// TwinCAT 3 PLC project PLC
// ProgramVersion: 3.1.4024.0
// libraries:
//   Tc2_Standard, * (Beckhoff Automation GmbH)
//   Tc2_System, * (Beckhoff Automation GmbH)
//   Tc3_Module, * (Beckhoff Automation GmbH)
// project tree:
//   / GlobalTextList.TcGTLO, PlcTask.TcTTO, Visualization Manager.TcVMO (not stored)
//   POUs/ MAIN.TcPOU
//   VISUs/ Visualization.TcVIS
// real-time tasks:
//   TASK PlcTask: cycle T#10ms, priority 20, ADS port 350

CONFIGURATION PLC
    RESOURCE PLC ON TwinCAT3
        TASK PlcTask(INTERVAL := T#10ms, PRIORITY := 20);
        PROGRAM MAIN WITH PlcTask : MAIN;
    END_RESOURCE
END_CONFIGURATION

// ---- POUs/MAIN.TcPOU
PROGRAM MAIN
VAR
	// push buttons
	StartPB: BOOL;
	StopPB: BOOL;
	ResetButton: BOOL;

	// sensors
	BottomLimitSwitch: BOOL;	
	ProxSwitch: BOOL;
	
	PistonLeftPos: BOOL;
	PistonRightPos: BOOL;
	
	// HW outputs
	
	ConveyorRun: BOOL;
	LifterUp: BOOL;
	LifterDown: BOOL;
	LifterStop: BOOL;
	
	PistonMoveLeft: BOOL;
	PistonMoveRight: BOOL;

	// Aux. objects
	rtBottomLS: R_TRIG;
	rtIndexPcb: R_TRIG;
	
	tondelayLifterUp: TON;
	tonDelay1sec: TON;
	
	rtPistonLeftReached: R_TRIG;
	ctuPistonLeftMovements: CTU;
END_VAR
VAR // added by the converter: edge detectors and wires of the graphical bodies
    _w1 : BOOL;
END_VAR

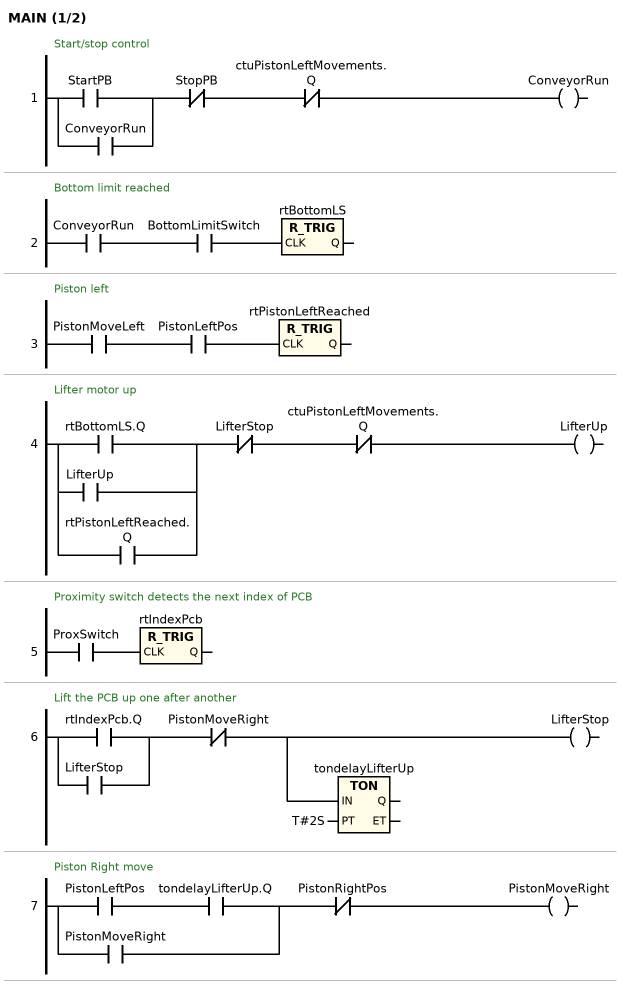
// NETWORK 1
// Start/stop control
ConveyorRun := (StartPB OR ConveyorRun) AND NOT StopPB AND NOT ctuPistonLeftMovements.Q;

// NETWORK 2
// Bottom limit reached
rtBottomLS(CLK := ConveyorRun AND BottomLimitSwitch); // R_TRIG

// NETWORK 3
// Piston left
rtPistonLeftReached(CLK := PistonMoveLeft AND PistonLeftPos); // R_TRIG

// NETWORK 4
// Lifter motor up
LifterUp := (rtBottomLS.Q OR LifterUp OR rtPistonLeftReached.Q) AND NOT LifterStop AND NOT ctuPistonLeftMovements.Q;

// NETWORK 5
// Proximity switch detects the next index of PCB
rtIndexPcb(CLK := ProxSwitch); // R_TRIG

// NETWORK 6
// Lift the PCB up one after another
_w1 := (rtIndexPcb.Q OR LifterStop) AND NOT PistonMoveRight;
LifterStop := _w1;
tondelayLifterUp(IN := _w1, PT := T#2S); // TON

// NETWORK 7
// Piston Right move
PistonMoveRight := (PistonLeftPos AND tondelayLifterUp.Q OR PistonMoveRight) AND NOT PistonRightPos;

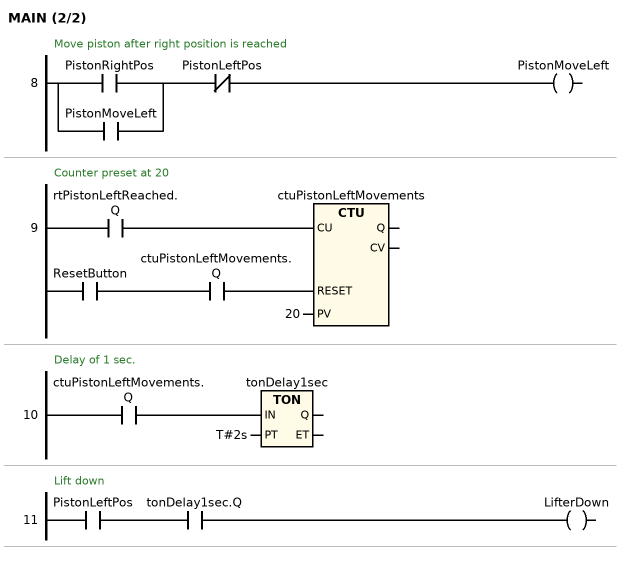
// NETWORK 8
// Move piston after right position is reached
PistonMoveLeft := (PistonRightPos OR PistonMoveLeft) AND NOT PistonLeftPos;

// NETWORK 9
// Counter preset at 20
ctuPistonLeftMovements(
    CU := rtPistonLeftReached.Q,
    RESET := ResetButton AND ctuPistonLeftMovements.Q,
    PV := 20); // CTU

// NETWORK 10
// Delay of 1 sec.
tonDelay1sec(IN := ctuPistonLeftMovements.Q, PT := T#2s); // TON

// NETWORK 11
// Lift down
LifterDown := PistonLeftPos AND tonDelay1sec.Q;

END_PROGRAM

// ---- GlobalTextList.TcGTLO
TEXTLIST GlobalTextList
  290 = 'Bottom LS'
  452 = 'Conveyor Run'
  528 = 'Lifter'
  534 = 'Piston Left Pos'
  221 = 'Piston Right Pos'
  535 = 'Prox. switch'
  58 = 'start PB'
  407 = 'stop PB'
  340 = 'stopPB'
END_TEXTLIST

// ---- VISUs/Visualization.TcVIS
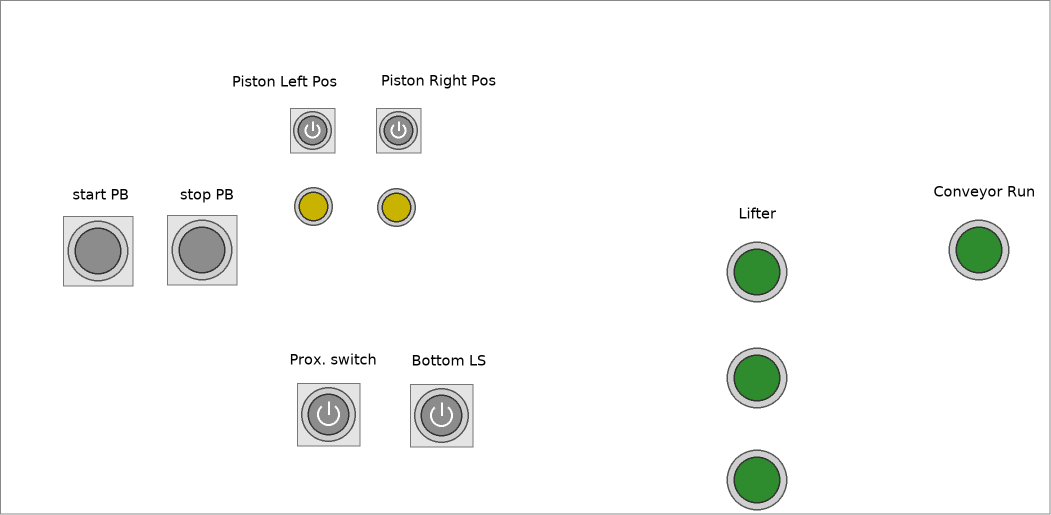
VISUALIZATION Visualization  // 1051x515
    PushSwitch (63,216 70x70), variable: MAIN.StartPB, behaviour: TAP, style: Switch-PushSwitch-Gray
    PushSwitch (167,215 70x70), variable: MAIN.StopPB, behaviour: TAP, style: Switch-PushSwitch-Gray
    PowerSwitch (297,381 63x67), variable: MAIN.ProxSwitch, behaviour: TOGGLE, style: Switch-PowerSwitch-Gray
    Lamp1 (944,215 70x70), variable: MAIN.ConveyorRun, style: Lamp-Lamp1-Green
    Lamp1 (722,237 70x70), variable: MAIN.LifterUp, style: Lamp-Lamp1-Green
    Lamp1 (722,343 70x70), variable: MAIN.LifterStop, style: Lamp-Lamp1-Green
    Label (50,174 102x41), "start PB"
    Label (156,174 102x41), "stop PB"
    Label (282,339 102x41), "Prox. switch"
    PowerSwitch (410,382 63x67), variable: MAIN.BottomLimitSwitch, behaviour: TOGGLE, style: Switch-PowerSwitch-Gray
    Label (398,340 102x41), "Bottom LS"
    PowerSwitch (290,103 45x55), variable: MAIN.PistonLeftPos, behaviour: TOGGLE, style: Switch-PowerSwitch-Gray
    PowerSwitch (376,103 45x55), variable: MAIN.PistonRightPos, behaviour: TOGGLE, style: Switch-PowerSwitch-Gray
    Label (222,61 125x41), "Piston Left Pos"
    Label (372,60 133x41), "Piston Right Pos"
    Label (918,171 133x41), "Conveyor Run"
    Lamp1 (722,445 70x70), variable: MAIN.LifterDown, style: Lamp-Lamp1-Green
    Label (691,193 133x41), "Lifter"
    Lamp1 (374,181 45x53), variable: MAIN.PistonMoveRight, style: Lamp-Lamp1-Yellow
    Lamp1 (291,180 45x53), variable: MAIN.PistonMoveLeft, style: Lamp-Lamp1-Yellow
END_VISUALIZATION
